FUNCTION_BLOCK Motor_Partida_Direta (* Composite Function Block Type *)
  (* Standard: 61499-2 *)
  (* Version 0.0, 15/01/2026, Schneider Electric, template *)
  PACKAGE Hidryco.HidrycoLib;
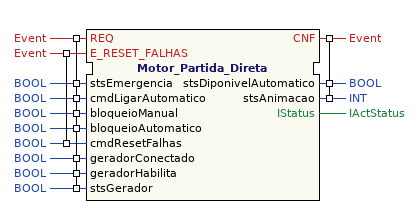
  EVENT_INPUT
    REQ WITH bloqueioManual, bloqueioAutomatico, cmdLigarAutomatico, geradorConectado, geradorHabilita, stsGerador, stsEmergencia;
    E_RESET_FALHAS WITH cmdResetFalhas;
  END_EVENT
  EVENT_OUTPUT
    CNF WITH stsDiponivelAutomatico, stsAnimacao;
  END_EVENT
  VAR_INPUT
    stsEmergencia : BOOL;
    cmdLigarAutomatico : BOOL;
    bloqueioManual : BOOL;
    bloqueioAutomatico : BOOL;
    cmdResetFalhas : BOOL;
    geradorConectado : BOOL;
    geradorHabilita : BOOL;
    stsGerador : BOOL;
  END_VAR
  VAR_OUTPUT
    stsDiponivelAutomatico : BOOL;
    stsAnimacao : INT;
  END_VAR
  PLUGS
    IStatus : IActStatus;
  END_PLUGS
  (* 0 - INITIALIZATION *)
  (* 1 - FUNCTIONAL INPUT INTERFACE *)
  (* 6 - OT-IT INTERFACE *)
  (* 2 - FUNCTIONAL OUTPUT INTERFACE *)
  (* 3 - FIELD INTERFACE *)
  (* 4 - CHILDREN *)
  (* 5 - LOGICS *)
  (* 4.A - TYPICALS *)
  (* 5.B - OPERATION MODE MANAGEMENT *)
  (* 5.C - INTERLOCKS MANAGEMENT *)
  (* 5.A - FUNCTIONAL BEHAVIORS *)
  (* 4.B- CHILDRENSS *)
  FBS
    IThis : Motor_Partida_Direta_HMI(QI := TRUE);
    SYMLINKMULTIVARDST1 : SYMLINKMULTIVARDST_65D63179E2618F5E(QI := TRUE, NAME1 := '$${PATH}stsFalhaComunicacao', NAME2 := '$${PATH}stsRemoto', NAME3 := '$${PATH}stsLocal', NAME4 := '$${PATH}stsLigado', NAME5 := '$${PATH}stsProtecao'); {SET_ATTRIBUTE(Configuration.GenericFBType.InterfaceParams, Runtime.System#I:=5;VALUE${I$}:BOOL,BOOL,BOOL,BOOL,BOOL)}
    SYMLINKMULTIVARSRC1 : SYMLINKMULTIVARSRC_277E97BEC1451D2C(NAME1 := '$${PATH}cmdAcionamento', NAME2 := '$${PATH}cmdReset'); {SET_ATTRIBUTE(Configuration.GenericFBType.InterfaceParams, Runtime.System#I:=2;VALUE${I$}:BOOL,BOOL)}
    plcStart1 : plcStart(Prio := 10);
  END_FBS
  EVENT_CONNECTIONS
    plcStart1.FIRST_INIT TO IThis.5A89AB6C3ADD5147;
    plcStart1.REDO_INIT TO IThis.5A89AB6C3ADD5147;
    IThis.34AE298E8667E33 TO IThis.18935C505C51E728;
    SYMLINKMULTIVARDST1.CNF TO IThis.9F1E8C85F66FE6FE;
    SYMLINKMULTIVARDST1.INITO TO SYMLINKMULTIVARSRC1.INIT;
    SYMLINKMULTIVARSRC1.INITO TO plcStart1.ACK_FIRST;
    E_RESET_FALHAS TO SYMLINKMULTIVARSRC1.REQ;
    SYMLINKMULTIVARDST1.CNF TO IStatus.14377629A1F197A9;
  END_CONNECTIONS
  DATA_CONNECTIONS
    SYMLINKMULTIVARDST1.VALUE2 TO IThis.DB7E989EF9FC4F63;
    SYMLINKMULTIVARDST1.VALUE5 TO IThis.C0C822B05EAB746F;
    cmdResetFalhas TO SYMLINKMULTIVARSRC1.VALUE2;
    SYMLINKMULTIVARDST1.VALUE4 TO IStatus.D41A46B14EF7208D;
  END_CONNECTIONS
END_FUNCTION_BLOCK
